PROGRAM Programma_test
VAR
END_VAR

END_PROGRAM

(* stored: Version 1.1.0.1, ProductVersion 3.1.4024.12
   POU Programma_test: Id {986bfd2d-1d24-4789-aa62-0d912b886579}, SpecialFunc None *)
